INTERFACE I_HE_SATT_FilterCombinationFinder


METHOD PUBLIC DetermineFilterCombinations
VAR_INPUT
    iFilterHolderSelector : I_HE_SATT_FilterHolderSelector;
    iFilterCombinationCollector : I_HE_SATT_FilterCombinationCollector;
END_VAR
END_METHOD


PROPERTY Status : REFERENCE TO ST_HE_SATT_Status
GET
END_GET
END_PROPERTY

END_INTERFACE

(* stored: Version 1.1.0.1
   Itf I_HE_SATT_FilterCombinationFinder: Id {66182892-49e1-4660-829e-cc3791522c27}
   Method DetermineFilterCombinations: Id {30980698-8e56-4802-a113-3fcf19607234}
   Property Status: Id {8a10b441-adf8-4ec2-a81d-e1818b464eda}
   Get Get: Id {85cedd68-a4d3-4e39-a89f-a637a8949ca8} *)
